(* IEC 61131-3 sources: volt/packages/volt-lsp-iec/test-corpus/bakon-nano/Device/Plc Logic/Application/Library Manager/SysTime, 3.5.9.0 (System), 5 files *)

(* ---- SVN_INFO_FLAGS.gvl ---- *)
VAR_GLOBAL
	XINCOMPLETE : BOOL := FALSE;
	XMODIFIED : BOOL := FALSE;
	XSWITCHED : BOOL := FALSE;
	XCLEAN : BOOL := TRUE;
END_VAR

(* ---- SVN_INFO_REVISIONS.gvl ---- *)
VAR_GLOBAL
	LIMINREVISION : LINT := LINT#6692;
	LIMAXREVISION : LINT := LINT#6692;
END_VAR

(* ---- SVN_INFO_SUMMARY.gvl ---- *)
VAR_GLOBAL
	SVERSIONSUMMARY : STRING(4) := '6692';
END_VAR

(* ---- SVN_INFO_SUMMARYW.gvl ---- *)
VAR_GLOBAL
	WSVERSIONSUMMARY : WSTRING(4) := "6692";
END_VAR

(* ---- SVN_INFO_URI.gvl ---- *)
VAR_GLOBAL
	WURL : WSTRING(82) := "svn://server04/LibrariesV3Source/branches/V3.5.9.0/System/SysLibs/SysTime/SysTime/";
END_VAR
